Universal Robots URScript: stringa_closer.script

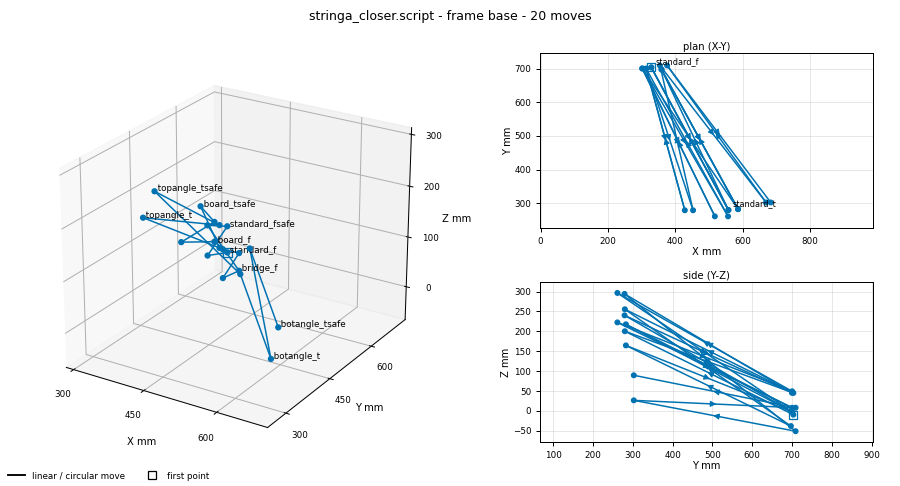
[picture p0: tool path of stringa_closer.script in frame base, 20 of 20 moves have a stored position in this frame; points joined in program order, loops and branches not executed]
def stringa_closer():
  global _hidden_verificationVariable=0
  set_safety_mode_transition_hardness(1)
  set_gravity([0.0, 0.0, 9.82])
  set_tool_communication(False, 115200, 0, 1, 1.5, 3.5)
  set_tool_output_mode(0)
  set_tool_digital_output_mode(0, 1)
  set_tool_digital_output_mode(1, 1)
  set_tool_voltage(0)
  set_target_payload(0.100000, [0.000000, 0.000000, 0.000000], [0.000033, 0.000033, 0.000033, 0.000000, 0.000000, 0.000000])
  set_standard_analog_input_domain(0, 1)
  set_standard_analog_input_domain(1, 1)
  set_tool_analog_input_domain(0, 1)
  set_tool_analog_input_domain(1, 1)
  set_analog_outputdomain(0, 0)
  set_analog_outputdomain(1, 0)
  set_input_actions_to_default()
  set_tcp(p[0.0,0.0,0.0,0.0,0.0,0.0])
  # begin: URCap Installation Node
  #   Source: External Control, 1.0.5, FZI Research Center for Information Technology
  #   Type: External Control
  # end: URCap Installation Node
  step_count_ee2dd8be_ac91_4144_8433_6be98217ca45 = 0.0
  thread Step_Counter_Thread_d86561a2_bd2e_4c9d_8836_359510afa219():
    while (True):
      step_count_ee2dd8be_ac91_4144_8433_6be98217ca45 = step_count_ee2dd8be_ac91_4144_8433_6be98217ca45 + 1.0
      sync()
    end
  end
  run Step_Counter_Thread_d86561a2_bd2e_4c9d_8836_359510afa219()
  global standard_f_p=p[.328964663774, .703229462539, -.009258082371, 1.501488908519, 2.294264795278, -1.521353569816]
  global standard_f_q=[-2.1784661451922815, -0.16920967519793706, 0.4420211950885218, -0.8301103276065369, -1.5967782179461878, -2.574190918599264]
  global standard_t_p=p[.557923990118, .279876247922, .200314083410, -1.446439182207, -2.240158754246, 1.575901583680]
  global standard_t_q=[-2.80978233018984, -0.8702692550471802, 1.2802026907550257, -1.004252867107727, -2.10295278230776, -2.944793764744894]
  global standard_fsafe_p=p[.328964663671, .703229462391, .045333550563, 1.501488908520, 2.294264795279, -1.521353569816]
  global standard_fsafe_q=[-2.17835236539009, -0.2402321061760091, 0.4473477656457767, -0.7644197264520631, -1.5968050732499393, -2.5743816886861204]
  global standard_tsafe_p=p[.557923989897, .279876247854, .255567513319, -1.446439179803, -2.240158755503, 1.575901584151]
  global standard_tsafe_q=[-2.809679111836697, -0.917689903288263, 1.2118107604793105, -0.8886419179810572, -2.103189450349886, -2.9451897721639853]
  global bridge_f_p=p[.359288490162, .697109874572, -.037989803078, -1.454279199729, -2.266388048891, 1.536760224005]
  global bridge_f_q=[-2.215261761342184, -0.04489179075274663, 0.25738269487489873, -0.7449875634959717, -1.5961187521563929, -2.6291380564319056]
  global bridge_t_p=p[.586461738590, .282502051645, .164701776524, -1.446439182239, -2.240158754244, 1.575901583647]
  global bridge_t_q=[-2.819451324470398, -0.7742163765849694, 1.2065189857476077, -1.029726718616942, -2.110909559167405, -2.950820149138915]
  global bridge_fsafe_p=p[.359288490131, .697109874486, -.001067425999, -1.454279200049, -2.266388049537, 1.536760222734]
  global bridge_fsafe_q=[-2.2151912998437444, -0.10803413529460393, 0.29411289248412825, -0.7185781000386653, -1.5960607083014056, -2.629240402831453]
  global bridge_tsafe_p=p[.586461738476, .282502051555, .217703154389, -1.446439181781, -2.240158754326, 1.575901583927]
  global bridge_tsafe_q=[-2.819344436212214, -0.8243593746292159, 1.1519376391450775, -0.9251965667014623, -2.1110940483836114, -2.9511965279821872]
  global board_f_p=p[.302077525790, .700121956010, .008096053708, 1.578563948242, 2.373499758638, -1.317137847045]
  global board_f_q=[-2.1552567142783587, -0.3371601412223937, 0.7412034669781562, -1.1085162439327227, -1.566591811570163, -2.551926211710005]
  global board_t_p=p[.517678248343, .261105329953, .222535084870, -1.474441172580, -2.232009306392, 1.513428520477]
  global board_t_q=[-2.8223379294024866, -0.9991956514171143, 1.434263054524557, -1.0614791077426453, -2.071507755910055, -2.9643142859088343]
  global board_fsafe_p=p[.302077525730, .700121956050, .049438367194, 1.578563955137, 2.373499757692, -1.317137839599]
  global board_fsafe_q=[-2.15516259694661, -0.3901991782063092, 0.7386730676661095, -1.0529463883408559, -1.5665922672270227, -2.5521122280433826]
  global board_tsafe_p=p[.556820561715, .261105329878, .296519711916, -1.474441171643, -2.232009306923, 1.513428520367]
  global board_tsafe_q=[-2.8404016543983843, -0.9782804252540034, 1.201472847702691, -0.8558833473401046, -2.0866822173097734, -2.9770976225380146]
  global topangle_f_p=p[.313606910374, .699665763876, -.001917473863, -1.688715616226, -1.887063138816, 1.664053082213]
  global topangle_f_q=[-2.193392578755514, -0.14644380033526616, 0.3925817648517054, -0.6567240518382569, -1.3763349691974085, -2.430572811757223]
  global topangle_t_p=p[.428451220547, .279140634606, .240209469554, -1.674748829325, -1.873859951039, 1.678075625066]
  global topangle_t_q=[-2.7635062376605433, -1.0948953193477173, 1.5453265349017542, -0.8615732950023194, -1.8955243269549769, -2.661124293004171]
  global topangle_fsafe_p=p[.313606910359, .699665763872, .045524839604, -1.688715651329, -1.887063157556, 1.664053021292]
  global topangle_fsafe_q=[-2.19329568295427, -0.2091532110992489, 0.39991926515343756, -0.601322059251924, -1.3763764976111652, -2.430729899103902]
  global topangle_tsafe_p=p[.452893533959, .279140634505, .294094096621, -1.674748829176, -1.873859951296, 1.678075624897]
  global topangle_tsafe_q=[-2.77830870578921, -1.0966032633912004, 1.400297356843998, -0.7170390438943288, -1.909550136237442, -2.6677407340689356]
  global botangle_f_p=p[.354749185881, .708893152215, -.050831555492, -1.033198855435, -2.489950727989, 1.270004512054]
  global botangle_f_q=[-2.2003896872149866, -0.10558863103900151, 0.4103601614581507, -0.981212930088379, -1.6054652372943323, -2.965921227131979]
  global botangle_t_p=p[.669656684572, .302367815533, .026684655516, -1.039222465315, -2.496995506148, 1.264917666173]
  global botangle_t_q=[-2.833883366970671, -0.4727017644621778, 1.0002373057657314, -1.3368387061026805, -2.0807023709782317, -3.4050013643523833]
  global botangle_fsafe_p=p[.375991499569, .708893151877, .008153071661, -1.033198855367, -2.489950728075, 1.270004512018]
  global botangle_fsafe_q=[-2.2199844149217816, -0.13595253071131808, 0.31946428876154, -0.8605220572607397, -1.6210376180921147, -2.9785547074625693]
  global botangle_tsafe_p=p[.683581126997, .302367815453, .089648590214, -1.039222444665, -2.496995494610, 1.264917705729]
  global botangle_tsafe_q=[-2.839018207845349, -0.5216170937585645, 0.9221434123972179, -1.212218527417897, -2.0844090481329527, -3.4098539460222916]
  while (True):
    $ 2 "Robot Program"
    $ 3 "MoveL"
    $ 4 "standard_f" "breakAfter"
    movel(standard_f_p, a=1.2, v=0.25)
    $ 5 "standard_t" "breakAfter"
    movel(standard_t_p, a=1.2, v=0.25)
    $ 6 "MoveL"
    $ 7 "standard_fsafe" "breakAfter"
    movel(standard_fsafe_p, a=1.2, v=0.25)
    $ 8 "standard_tsafe" "breakAfter"
    movel(standard_tsafe_p, a=1.2, v=0.25)
    $ 9 "MoveL"
    $ 10 "bridge_f" "breakAfter"
    movel(bridge_f_p, a=1.2, v=0.25)
    $ 11 "bridge_t" "breakAfter"
    movel(bridge_t_p, a=1.2, v=0.25)
    $ 12 "MoveL"
    $ 13 "bridge_fsafe" "breakAfter"
    movel(bridge_fsafe_p, a=1.2, v=0.25)
    $ 14 "bridge_tsafe" "breakAfter"
    movel(bridge_tsafe_p, a=1.2, v=0.25)
    $ 15 "MoveL"
    $ 16 "board_f" "breakAfter"
    movel(board_f_p, a=1.2, v=0.25)
    $ 17 "board_t" "breakAfter"
    movel(board_t_p, a=1.2, v=0.25)
    $ 18 "MoveL"
    $ 19 "board_fsafe" "breakAfter"
    movel(board_fsafe_p, a=1.2, v=0.25)
    $ 20 "board_tsafe" "breakAfter"
    movel(board_tsafe_p, a=1.2, v=0.25)
    $ 21 "MoveL"
    $ 22 "topangle_f" "breakAfter"
    movel(topangle_f_p, a=1.2, v=0.25)
    $ 23 "topangle_t" "breakAfter"
    movel(topangle_t_p, a=1.2, v=0.25)
    $ 24 "MoveL"
    $ 25 "topangle_fsafe" "breakAfter"
    movel(topangle_fsafe_p, a=1.2, v=0.25)
    $ 26 "topangle_tsafe" "breakAfter"
    movel(topangle_tsafe_p, a=1.2, v=0.25)
    $ 27 "MoveL"
    $ 28 "botangle_f" "breakAfter"
    movel(botangle_f_p, a=1.2, v=0.25)
    $ 29 "botangle_t" "breakAfter"
    movel(botangle_t_p, a=1.2, v=0.25)
    $ 30 "MoveL"
    $ 31 "botangle_fsafe" "breakAfter"
    movel(botangle_fsafe_p, a=1.2, v=0.25)
    $ 32 "botangle_tsafe" "breakAfter"
    movel(botangle_tsafe_p, a=1.2, v=0.25)
  end
end
